# EPICS autosave request: measCompApp/Db/C9513_counter_settings.req
$(P)$(R)GateControl
$(P)$(R)CounterEdge
$(P)$(R)CountSource
$(P)$(R)SpecialGate
$(P)$(R)ReloadSource
$(P)$(R)RecycleMode
$(P)$(R)BCDMode
$(P)$(R)CountDirection
$(P)$(R)OutputControl
$(P)$(R)LoadReg
$(P)$(R)HoldReg
$(P)$(R)PollCounter
